TYPE DUT :
STRUCT
END_STRUCT
END_TYPE

(* stored: Version 1.1.0.1, ProductVersion 3.1.4024.12
   DUT DUT: Id {82a97e48-6624-4814-87e8-1866e8ae5f8e} *)
